# EPICS substitutions: elioApp/Db/EL1124.substitutions
file EL1124.template { pattern
{ CHAN	}
{ 1	}
{ 2	}
{ 3	}
{ 4	}
}
